PROGRAM a6_Lecture_InterCom
VAR
	Cons_Temp_Eau_General: REAL;
END_VAR

(**********************************************Gestion lecture inter com*)
MES_Temp_Eau_Mitige_General := Tab_Com_Receive[0];
Cons_Temp_Eau_General		:= Tab_Com_Receive[1];

END_PROGRAM

(* stored: Version 1.1.0.1, ProductVersion 3.1.4024.15
   POU a6_Lecture_InterCom: Id {567fc0bc-06c9-411d-994a-f073a4899aa5}, SpecialFunc None *)
